// TwinCAT 3 PLC project ABDriveCom
// ProgramVersion: 3.1.4023.0
// libraries:
//   Tc2_MC2, * (Beckhoff Automation GmbH)
//   Tc2_Standard, * (Beckhoff Automation GmbH)
//   Tc2_System, * (Beckhoff Automation GmbH)
//   Tc3_Module, * (Beckhoff Automation GmbH)
//   VisuSymbols,3.5.10.0,System
// project tree:
//   / GlobalTextList.TcGTLO, PlcTask.TcTTO, Visualization Manager.TcVMO (not stored)
//   GVLs/ GVL.TcGVL
//   POUs/ MAIN.TcPOU, Sequence.TcPOU
//   VISUs/ Visualization.TcVIS, VisualizationTwinCAT.TcVIS
// real-time tasks:
//   TASK Task 4: cycle T#1ms, priority 1, ADS port 301
//   TASK PlcTask: cycle T#10ms, priority 20, ADS port 350
// motion (NC):
//   TASK NC-Task 1 SAF: cycle T#2ms, priority 4, ADS port 501
//   TASK NC-Task 1 SVB: cycle T#10ms, priority 8, ADS port 511
//   AXIS Axis 1 (id 1)
//     Dynamic: Acceleration=13141.3, Deceleration=13141.3, Jerk=39423.8
//     Velo: RefSearch=87.6085248, RefSync=87.6085248, SlowManual=438.042624, FastManual=2628.255744, Fast=8760.85248, Maximum=8760.85
//     OtherSettings: AllowMotionCmdToSlave=true
//     encoder EncType=19
//       EncPara: ScaleFactorNumerator=104.8576, ScaleFactorDenominator=1048576, MaxCount=#xffffffff
//     drive DrvType=16
//       DrvPara: MaxCount=#xffffffff, DriveControlDWord=#x00020000
//         Analog: VeloReferenz=9636.937728, VeloScale=32, TorqueSetpointScale=10, ScaleFactorActTorque=0.1
//         TimeComp: TaskDelayCycles=1
//     controller CtrType=1
//       CtrPara: PriorControlFactor=1
//         PosDiffControl: Range=10, Time=1
//         PID: PosKp=8
//         Observer: BandWidth=20
// I/O:
//   DEVICE Device 2 (TC3 EIP Scanner), AmsNetId 5.109.28.196.3.1
//     Box 7 (EtherNet/IP Slave (generic)) // <INFO> </INFO> <EDS> C:\TwinCAT\3.1\Config\Io\EtherNetIP\ </EDS>
//     Box 8 (Producer Object List)
//   DEVICE Device 1 (EtherCAT), AmsNetId 5.109.28.196.2.1
//     Term 1 (EK1200) [EK1200-5000 EtherCAT Power supply (2A E-Bus)]
//       Term 3 (EL6910) [EL6910, TwinSAFE PLC]
//       Term 4 (EL1904) [EL1904, 4 Ch. Safety Input 24V, TwinSAFE]
//         modules: Module 1 (FSOES)
//       Term 5 (EL7201-0010) [EL7201-0010 1Ch. MDP742 Servo motor output stage with OCT (50V, 4A)]
//       Term 6 (EK1110) [EK1110 EtherCAT extension]
//   DEVICE Device 5 (USB)
//     Box 1 (CX2100 Power Supply)
// variable links:
//   NC-Task 1 SAF/Axes/Axis 1 <-> Device 1 (EtherCAT)/Term 1 (EK1200)/Term 5 (EL7201-0010)
//     Drive/Inputs/In/nDcOutputTime <-> InfoData/DcOutputShift
//     Drive/Inputs/In/nState1 <-> DRV Statusword/Statusword
//     Drive/Inputs/In/nState2 <-> DRV Statusword/Statusword @bit 8
//     Drive/Inputs/In/nState4 @bit 1 <-> WcState/InputToggle
//     Drive/Inputs/In/nState4 <-> WcState/WcState
//     Drive/Outputs/Out/nCtrl1 <-> DRV Controlword/Controlword
//     Drive/Outputs/Out/nCtrl2 <-> DRV Controlword/Controlword @bit 8
//     Drive/Outputs/Out/nDataOut2 <-> DRV Target velocity/Target velocity
//     Enc/Inputs/In/nDataIn1 <-> FB Position/Position
//     Enc/Inputs/In/nDcInputTime <-> InfoData/DcInputShift
//     Enc/Inputs/In/nState4 @bit 1 <-> WcState/InputToggle
//     Enc/Inputs/In/nState4 <-> WcState/WcState
//   ABDriveCom/ABDriveCom Instance <-> Device 2 (TC3 EIP Scanner)
//     PlcTask Inputs/MAIN.AB_Connected <-> Inputs/DevState
//   ABDriveCom/ABDriveCom Instance <-> Device 2 (TC3 EIP Scanner)/Box 7 (EtherNet/IP Slave (generic))
//     PlcTask Inputs/GVL.ABIN1 <-> AB DINT IN/Inputs/TwinCAT_IN[0]
//     PlcTask Inputs/GVL.ABIN2 <-> AB DINT IN/Inputs/TwinCAT_IN[1]
//     PlcTask Inputs/MAIN.ProgramStep <-> AB DINT IN/Inputs/TwinCAT_IN[2]
//   ABDriveCom/ABDriveCom Instance <-> Device 2 (TC3 EIP Scanner)/Box 8 (Producer Object List)
//     PlcTask Outputs/GVL.ABOUT2 <-> Producer 2 (Output)/Outputs/TwinCAT_OUT[1]
//     PlcTask Outputs/GVL.ABOUT3 <-> Producer 2 (Output)/Outputs/TwinCAT_OUT[2]
//     PlcTask Outputs/MAIN.TwinCAT_StartProgram <-> Producer 2 (Output)/Outputs/TwinCAT_OUT[0] @bit 7
//     PlcTask Outputs/MAIN.TwinCAT_bEnable <-> Producer 2 (Output)/Outputs/TwinCAT_OUT[0] @bit 1
//     PlcTask Outputs/MAIN.TwinCAT_bReset <-> Producer 2 (Output)/Outputs/TwinCAT_OUT[0] @bit 2
//     PlcTask Outputs/MAIN.TwinCAT_jogBack <-> Producer 2 (Output)/Outputs/TwinCAT_OUT[0] @bit 4
//     PlcTask Outputs/MAIN.TwinCAT_jogFwd <-> Producer 2 (Output)/Outputs/TwinCAT_OUT[0] @bit 3
//   ABDriveCom/ABDriveCom Instance <-> Device 5 (USB)/Box 1 (CX2100 Power Supply)
//     PlcTask Inputs/MAIN.ContollerStart <-> DIS Inputs/Status/Enter
//   ABDriveCom/ABDriveCom Instance <-> NC-Task 1 SAF/Axes/Axis 1
//     PlcTask Inputs/MAIN.Axis1.NcToPlc <-> Outputs/ToPlc
//     PlcTask Outputs/MAIN.Axis1.PlcToNc <-> Inputs/FromPlc

CONFIGURATION ABDriveCom
    RESOURCE PLC ON TwinCAT3
        TASK PlcTask(INTERVAL := T#10ms, PRIORITY := 20);
        PROGRAM MAIN WITH PlcTask : MAIN;
    END_RESOURCE
END_CONFIGURATION

// ---- GVLs/GVL.TcGVL
{attribute 'qualified_only'}
VAR_GLOBAL
	ABIN1 AT %I* :DINT;
	ABIN2 AT %I* :DINT;
	ABOUT1 AT %Q* :DINT;
	ABOUT2 AT %Q* :DINT;
	ABOUT3 AT %Q* :DINT;
END_VAR

// ---- POUs/MAIN.TcPOU
PROGRAM MAIN
VAR
  Axis1 : AXIS_REF;
  Axis1Power 	: MC_Power;
  Axis1Move		: MC_MoveAbsolute;
  Axis1Jog		: MC_Jog;
  Axis1Reset	: MC_Reset;
  Axis1Home		: MC_Home;
  
  
	bABEnable		AT	%I* : BOOL;
	bABExecuteMove AT %I*: BOOL;
	bABJogForward		AT	%I* : BOOL;
	bABJogBackward	 AT	%I* : BOOL;
	bABAxisReset	 AT	%I* : BOOL;
	bABResetDone	AT %Q*: BOOL;
	bABMoveDone AT %Q*: BOOL;
	bABError AT %Q*: BOOL;
	
	ProgramStep AT %I* :DINT;
	
	TwinCAT_bEnable	AT %Q*: BOOL;
	TwinCAT_bReset AT %Q*: BOOL;
	TwinCAT_jogFwd AT %Q*: BOOL;
	TwinCAT_jogBack AT %Q*: BOOL;
	TwinCAT_StartProgram AT %Q*: BOOL;
	
	AB_Connected AT %I* :UINT;
	DriveErrorCode : UDINT ; ///	AT %I* :UDINT;

	LinkError: BOOL;
	bExecuteHome: BOOL;
	
	bEnable			 : BOOL;
	bExecuteMove	 : BOOL;
	bJogForward		 : BOOL;
	bJogBackward	 : BOOL;
	bAxisReset	 	 : BOOL;
	bResetDone		 : BOOL;
	bMoveDone 		 : BOOL;
	bError 			 : BOOL;
	
	Position		 : LREAL;
	Velocity		 : LREAL;

	StartSeq			: BOOL;
	Sequence 		: Sequence;
	bRunContinuous	: BOOL;
	bJogEnable: BOOL;
	bJogReset: BOOL;
	
	ContollerStart AT %I* : BOOL;
	
	
	//SAFETY TEST
	ErrorAck AT %Q* : BOOL;
	Reset	AT %Q* : BOOL;
	RUN		AT %Q* : BOOL;
	Test	AT %Q* : BOOL;
	Test2	AT %Q* : BOOL;
END_VAR

Axis1Power(
	Axis:= Axis1, 
	Enable:= bABEnable OR bEnable OR bJogEnable, 
	Enable_Positive:= bABEnable OR bEnable OR bJogEnable, 
	Enable_Negative:= bABEnable OR bEnable OR bJogEnable, 
	Override:= 100, 
	BufferMode:= , 
	Options:= , 
	Status=> , 
	Busy=> , 
	Active=> , 
	Error=> bError, 
	ErrorID=> DriveErrorCode);
	
Axis1Jog(
	Axis:= Axis1, 
	JogForward:= bABJogForward OR bJogForward, 
	JogBackwards:= bABJogBackward OR bJogBackward, 
	Mode:= E_JogMode.MC_JOGMODE_STANDARD_SLOW, 
	Position:= , 
	Velocity:= 100, 
	Acceleration:= 10000, 
	Deceleration:= 10000, 
	Jerk:= 10000, 
	Done=> , 
	Busy=> , 
	Active=> , 
	CommandAborted=> , 
	Error=> , 
	ErrorID=> );

Axis1Move(
	Axis:= Axis1, 
	Execute:= bABExecuteMove OR bExecuteMove, 
	Position:= Position, 
	Velocity:= Velocity, 
	Acceleration:= 5000, 
	Deceleration:= 5000, 
	Jerk:= 10000, 
	BufferMode:= , 
	Options:= , 
	Done=> bMoveDone, 
	Busy=> , 
	Active=> , 
	CommandAborted=> , 
	Error=> , 
	ErrorID=> );	
	
Axis1Reset(
	Axis:= Axis1, 
	Execute:= bABAxisReset OR bAxisReset OR bJogReset, 
	Done=> bResetDone, 
	Busy=> , 
	Error=> , 
	ErrorID=> );	
	
Axis1Home(
	Axis:= Axis1, 
	Execute:= bExecuteHome, 
	Position:= 0, 
	HomingMode:= MC_Direct, 
	BufferMode:= , 
	Options:= , 
	bCalibrationCam:= , 
	Done=> , 
	Busy=> , 
	Active=> , 
	CommandAborted=> , 
	Error=> , 
	ErrorID=> );	
	
IF AB_Connected >= 1 THEN
	LinkError := TRUE;
ELSE
	LinkError := FALSE;	
END_IF	

Sequence(StartSeq := StartSeq,
		 bEnable => bEnable,
		 bReset => bAxisReset,
		 Position => Position,
		 Velocity => Velocity,
		 ExecuteMove => bExecuteMove,
		bRunContinuous := bRunContinuous);
		 
IF ContollerStart THEN
	StartSeq := TRUE;
END_IF

END_PROGRAM

// ---- POUs/Sequence.TcPOU
FUNCTION_BLOCK Sequence

VAR
	Seq : INT;
	PositionInfo : ARRAY [0..9] OF LREAL; 
	VelocityInfo : ARRAY [0..9] OF LREAL;	
	i : INT;
END_VAR

VAR_OUTPUT
	bEnable	: BOOL;
	bReset	: BOOL;
	Position : LREAL;
	Velocity : LREAL;
	ExecuteMove : BOOL;
END_VAR

VAR_IN_OUT
	StartSeq : BOOL;
	bRunContinuous : BOOL;
END_VAR

MAIN.Axis1.ReadStatus();

PositionInfo[0] := 1000.0;		velocityInfo[0] := 5000.0;  
PositionInfo[1] := 	  0.0;		velocityInfo[1] := 1000.0;
PositionInfo[2] := 2000.0;		velocityInfo[2] := 600.0;
PositionInfo[3] := 1500.0;		velocityInfo[3] := 100.0;
PositionInfo[4] :=  -50.1;		velocityInfo[4] := 5000.0;
PositionInfo[5] := -950.0;		velocityInfo[5] := 5000.0;
PositionInfo[6] :=  500.0;		velocityInfo[6] := 2000.0;
PositionInfo[7] :=    5.2;		velocityInfo[7] := 5000.0;
PositionInfo[8] := -525.7;		velocityInfo[8] := 500.0;
PositionInfo[9] :=   45.5;		velocityInfo[9] := 1000.0;

CASE Seq OF 
	0:
		IF StartSeq THEN
			Seq := 1;
		END_IF
		
	1:
		bEnable := TRUE;
		IF MAIN.Axis1Power.Active THEN
			Seq := 5;
		END_IF
	
	5: 
		bReset := TRUE;
		IF MAIN.Axis1Reset.Done THEN
			bReset := FALSE;
			Seq := 10;
		END_IF
	
	10:
		Position := PositionInfo[i];
		Velocity := VelocityInfo[i];
		IF MAIN.Axis1.Status.Operational THEN
			ExecuteMove := TRUE;
			Seq := 15;
		END_IF
		
		
	15:
		IF MAIN.Axis1Move.Done THEN
			ExecuteMove := FALSE;
			Seq := 20;
		ELSIF MAIN.Axis1.Status.Error THEN
			ExecuteMove := FALSE;
			StartSeq := FALSE;	
			Seq := 0;
		END_IF
	
	20:
		i := i+1;
		
		IF i < 10 THEN
			Seq := 10;
		ELSIF i > 10 AND NOT bRunContinuous THEN
			i := 0;	
			Seq := 0;
			StartSeq := FALSE;
			bEnable := FALSE;
		ELSIF i > 10 AND bRunContinuous THEN
			i := 0;
			Seq := 10;
		END_IF	
END_CASE

END_FUNCTION_BLOCK

// ---- GlobalTextList.TcGTLO
TEXTLIST GlobalTextList
  17 = '%'
  384 = '%d'
  360 = '%i'
  245 = '%r'
  571 = '%s'
  128 = 'Axis Actual Position'
  130 = 'Axis Error Code'
  75 = 'Enable'
  359 = 'Ethernet/IP Communication'
  244 = 'JogBack'
  475 = 'JogFwd'
  151 = 'Program Loop'
  992 = 'Program Step'
  445 = 'Reset'
  215 = 'Run Program'
END_TEXTLIST

// ---- VISUs/Visualization.TcVIS
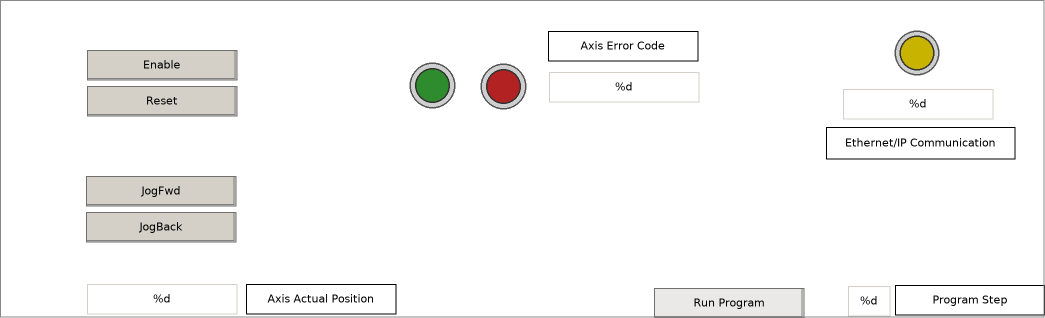
VISUALIZATION Visualization  // 1045x318
    Button (86,176 150x30), "JogFwd"
        OnMouseDown: toggle MAIN.TwinCAT_jogFwd
        OnMouseUp: toggle MAIN.TwinCAT_jogFwd
    Button (86,212 150x30), "JogBack"
        OnMouseDown: toggle MAIN.TwinCAT_jogBack
        OnMouseUp: toggle MAIN.TwinCAT_jogBack
    Lamp1 (406,57 53x57), variable: MAIN.bEnable, style: Lamp-Lamp1-Green
    Lamp1 (477,59 53x55), variable: MAIN.bError, style: Lamp-Lamp1-Red
    Button (87,50 150x30), "Enable"
        OnMouseDown: toggle MAIN.TwinCAT_bEnable
    Button (87,86 150x30), "Reset"
        OnMouseDown: toggle MAIN.TwinCAT_bReset
        OnMouseUp: toggle MAIN.TwinCAT_bReset
    Lamp1 (891,27 52x52), variable: MAIN.LinkError, style: Lamp-Lamp1-Yellow
    Textfield (843,89 150x30), "%d", text variable: MAIN.AB_Connected
    Textfield (549,72 150x30), "%d", text variable: MAIN.DriveErrorCode
    Textfield (87,284 150x30), "%d", text variable: MAIN.Axis1.NcToPlc.ActPos
    Button (654,288 150x30), "Run Program", colour toggle: MAIN.TwinCAT_StartProgram
        OnMouseDown: toggle MAIN.TwinCAT_StartProgram
    Textfield (848,286 42x30), "%d", text variable: MAIN.ProgramStep
    Rectangle (548,31 150x30), "Axis Error Code"
    Rectangle (826,127 189x32), "Ethernet/IP Communication"
    Rectangle (246,284 150x30), "Axis Actual Position"
    Rectangle (895,285 150x30), "Program Step"
END_VISUALIZATION

// ---- VISUs/VisualizationTwinCAT.TcVIS
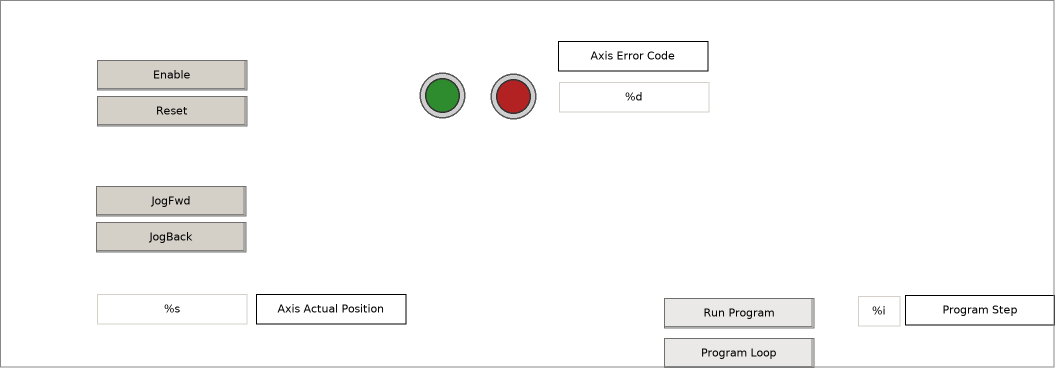
VISUALIZATION VisualizationTwinCAT  // 1055x368
    Button (96,186 150x30), "JogFwd"
        OnMouseDown: toggle MAIN.bJogForward
        OnMouseUp: toggle MAIN.bJogForward
    Button (96,222 150x30), "JogBack"
        OnMouseDown: toggle MAIN.bJogBackward
        OnMouseUp: toggle MAIN.bJogBackward
    Lamp1 (416,67 53x57), variable: MAIN.Axis1.Status.Operational, style: Lamp-Lamp1-Green
    Lamp1 (487,69 53x55), variable: MAIN.bError, style: Lamp-Lamp1-Red
    Button (97,60 150x30), "Enable"
        OnMouseDown: toggle MAIN.bJogEnable
    Button (97,96 150x30), "Reset"
        OnMouseDown: toggle MAIN.bJogReset
        OnMouseUp: toggle MAIN.bJogReset
    Textfield (559,82 150x30), "%d", text variable: MAIN.DriveErrorCode
    Textfield (97,294 150x30), "%s", text variable: MAIN.Axis1.NcToPlc.ActPos
    Button (664,298 150x30), "Run Program", colour toggle: MAIN.StartSeq
        OnMouseDown: toggle MAIN.StartSeq
    Textfield (858,296 42x30), "%i", text variable: MAIN.Sequence.i
    Rectangle (558,41 150x30), "Axis Error Code"
    Rectangle (256,294 150x30), "Axis Actual Position"
    Rectangle (905,295 150x30), "Program Step"
    Button (664,338 150x30), "Program Loop", colour toggle: MAIN.bRunContinuous, invisible if: NOT MAIN.StartSeq
        OnMouseDown: toggle MAIN.bRunContinuous
END_VISUALIZATION
